// Provies interface to properties required for file access
INTERFACE I_FileProperties

// Gets or set file properties.
PROPERTY File : REFERENCE TO ST_FileInfo
GET
END_GET
END_PROPERTY

END_INTERFACE

(* stored: Version 1.1.0.1, ProductVersion 3.1.4024.14
   Itf I_FileProperties: Id {43aa2010-3609-05d0-1056-3d643eef0756}
   Property File: Id {824aac20-18df-01b9-0ec6-ca8d100bf84d}
   Get Get: Id {c78d7bcc-1184-0016-387d-e1a0ed61f88e} *)
